Universal Robots PolyScope program: finalcoffee19-05-03.urp

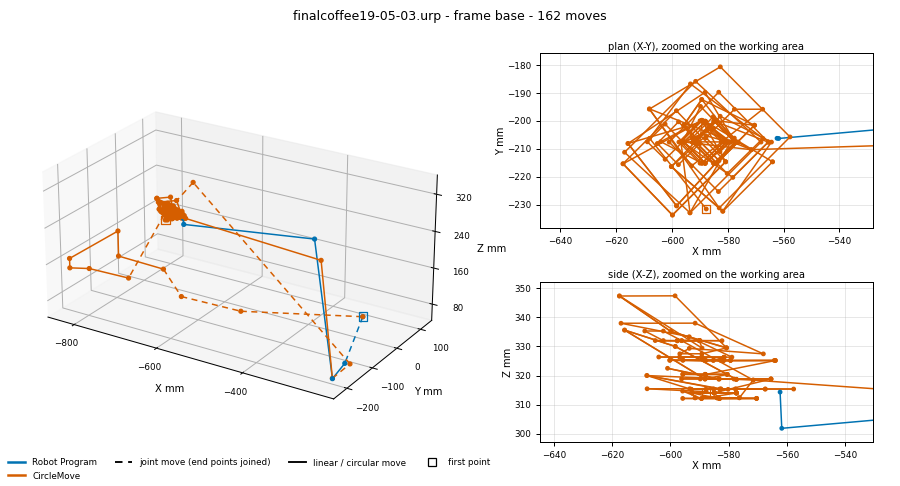
[picture p0: tool path of finalcoffee19-05-03.urp in frame base, 162 of 162 moves have a stored position in this frame; points joined in program order, loops and branches not executed]
Program finalcoffee19-05-03 (createdIn=3.3.3.292 lastSavedIn=3.3.3.292 directory=/programs/usbdisk_0 installation=default robotSerialNumber=2016353566)
Calibrated DH parameters: a=[0.000241, -0.028217, -0.285075, -0.000076, 0.000104, 0]; d=[0.089155, 574.834368, -342.811798, -231.912434, 0.094822, 0.082605]; alpha=[1.570306, 0.000738, 0.001161, 1.569845, -1.570892, 0]; deltaTheta=[0.000027, 1.504353, -0.747309, -0.757122, 0.000051, -0.000036]
Robot Program (runOnlyOnce=true motionType=MoveJ speed=1.047198 acceleration=1.396263 recalculateMotions=false)
  URCap com.ur.urcap.OnRobot.HelloWorldNode data=depthCompensate = false
    | width = 40
    | name = RG2(40)
    | force = 40
  MoveJ speed 20 deg/s, acceleration 30 deg/s^2 (recalculateMotions=false)
    Waypoint Waypoint_11: TCP in base x=-274.743 y=-2.169 z=93.833 mm, rx=1.4578 ry=-0.5495 rz=0.5386 rad; joints [-61.662, -71.825, 125.124, -50.852, -60.403, 38.941] deg; flange x=-270.843 y=184.262 z=86.813 mm, rx=1.4577 ry=-0.5495 rz=0.5386 rad
    Waypoint Waypoint_24: TCP in base x=-231.12 y=-150.401 z=66.269 mm, rx=0.5942 ry=1.8381 rz=-1.9212 rad; joints [-53.372, -80.21, 145.778, -62.89, -52.13, 33.023] deg; flange x=-227.221 y=36.081 z=59.238 mm, rx=1.4762 ry=-0.4771 rz=0.463 rad
  MoveP speed 76.2 mm/s, acceleration 1198.88 mm/s^2 (blendRadius=0.025 recalculateMotions=false) feature=Base
    Waypoint Waypoint_10: TCP in base x=-226.514 y=-206.056 z=58.912 mm, rx=0.3512 ry=2.0783 rz=-2.0466 rad; joints [-45.775, -85.681, 150.207, -66.123, -44.48, 19.129] deg; flange x=-222.338 y=-13.96 z=62.51 mm, rx=1.5718 ry=-0.2656 rz=0.2272 rad
  URCap com.ur.urcap.OnRobot.HelloWorldNode data=depthCompensate = false
    | width = 0
    | name = RG2(0)
    | force = 40
  URCap com.ur.urcap.OnRobot.TCPNode data=x = 5.6843418860808015E-14
    | y = -5.6843418860808015E-14
    | z = -2.5579538487363607E-13
    | rx = 0.0
    | ry = 5.551115123125783E-17
    | rz = 5.551115123125783E-17
    | xS = 0.0
    | yS = 0.0
    | zS = 0.0
    | rxS = 0.0
    | ryS = 0.0
    | rzS = 0.0
    | width = 40
    | tcpType = true
    | measuredWidthEnable = true
    | slaveSelected = false
    | TCP = TCP RG2()
  MoveL speed 76.2 mm/s, acceleration 254 mm/s^2 (recalculateMotions=false) feature=Base
    Waypoint wp_up: TCP in base x=-284.404 y=-181.482 z=326.495 mm, rx=0.3512 ry=2.0781 rz=-2.0466 rad; joints [-39.61, -106.093, 116.533, -12.17, -38.344, 19.314] deg; flange x=-280.343 y=5.056 z=329.988 mm, rx=1.5717 ry=-0.2657 rz=0.2273 rad
    Waypoint cup_center: TCP in base x=-561.773 y=-206.265 z=301.908 mm, rx=0.3623 ry=2.0424 rz=-1.9951 rad; joints [-18.068, -66.655, 77.97, -15.065, -18.801, 24.438] deg; flange x=-564.357 y=-14.16 z=305.939 mm, rx=1.5749 ry=-0.2793 rz=0.2941 rad
  MoveP speed 38.1 mm/s, acceleration 7.62 mm/s^2 (blendRadius=0.0127 recalculateMotions=false) feature=Base
    Waypoint cent_35: motionParameters(blendRadius=0.011); TCP in base x=-562.353 y=-206.199 z=314.344 mm, rx=0.5423 ry=1.9235 rz=-1.8764 rad; joints [-18.058, -66.887, 76.46, -13.315, -18.791, 35.8] deg; flange x=-564.912 y=-14.083 z=318.336 mm, rx=1.5494 ry=-0.4367 rz=0.4479 rad
    CircleMove
      Waypoint Waypoint_14: motionParameters(blendRadius=0.018); TCP in base x=-587.687 y=-231.512 z=314.467 mm, rx=0.5306 ry=1.932 rz=-1.8849 rad; joints [-14.904, -63.855, 72.029, -12.661, -15.633, 35.8] deg; flange x=-590.209 y=-39.4 z=318.513 mm, rx=1.5515 ry=-0.4261 rz=0.4373 rad
      Waypoint deg_left_36: motionParameters(blendRadius=0.013); TCP in base x=-607.977 y=-206.219 z=315.477 mm, rx=0.5411 ry=1.9244 rz=-1.8774 rad; joints [-16.716, -60.481, 66.783, -10.318, -17.442, 36.007] deg; flange x=-610.544 y=-14.142 z=319.49 mm, rx=1.5496 ry=-0.4357 rz=0.4467 rad
  MoveP speed 25.4 mm/s, acceleration 76.2 mm/s^2 (blendRadius=0.00635 recalculateMotions=false) feature=Base
    CircleMove
      Waypoint Waypoint_120: motionParameters(blendRadius=0.011); TCP in base x=-593.35 y=-186.719 z=315.478 mm, rx=0.5524 ry=1.9162 rz=-1.8691 rad; joints [-18.922, -62.136, 69.295, -10.741, -19.654, 36.3] deg; flange x=-595.922 y=5.421 z=319.508 mm, rx=1.5475 ry=-0.446 rz=0.457 rad
      Waypoint Waypoint_121: motionParameters(blendRadius=0.006); TCP in base x=-567.406 y=-206.241 z=315.399 mm, rx=0.5493 ry=1.9185 rz=-1.8715 rad; joints [-17.897, -66.224, 75.343, -12.894, -18.625, 36.3] deg; flange x=-569.935 y=-14.123 z=319.455 mm, rx=1.5481 ry=-0.4432 rz=0.4541 rad
    CircleMove
      Waypoint Waypoint_122: motionParameters(blendRadius=0.01); TCP in base x=-580.202 y=-218.815 z=315.281 mm, rx=0.5491 ry=1.9188 rz=-1.8724 rad; joints [-16.313, -64.705, 73.156, -12.546, -17.023, 36.581] deg; flange x=-582.655 y=-26.726 z=319.337 mm, rx=1.548 ry=-0.4427 rz=0.4531 rad
      Waypoint Waypoint_123: motionParameters(blendRadius=0.006); TCP in base x=-592.797 y=-206.153 z=315.297 mm, rx=0.5517 ry=1.9167 rz=-1.87 rad; joints [-17.153, -62.662, 70.126, -11.364, -17.868, 36.6] deg; flange x=-595.328 y=-13.997 z=319.293 mm, rx=1.5474 ry=-0.4457 rz=0.4562 rad
    CircleMove
      Waypoint Waypoint_124: motionParameters(blendRadius=0.003); TCP in base x=-585.199 y=-198.492 z=315.45 mm, rx=0.5527 ry=1.916 rz=-1.869 rad; joints [-18.086, -63.573, 71.462, -11.621, -18.81, 36.485] deg; flange x=-587.756 y=-6.367 z=319.434 mm, rx=1.5474 ry=-0.4464 rz=0.4572 rad
      Waypoint Waypoint_125: motionParameters(blendRadius=0.003); TCP in base x=-577.639 y=-206.134 z=315.376 mm, rx=0.5537 ry=1.9154 rz=-1.8684 rad; joints [-17.596, -64.801, 73.285, -12.319, -18.315, 36.654] deg; flange x=-580.185 y=-13.996 z=319.379 mm, rx=1.5472 ry=-0.4474 rz=0.4579 rad
    MoveP speed 25.4 mm/s, acceleration 25.4 mm/s^2 (blendRadius=0.00508 recalculateMotions=false) feature=Base
      CircleMove
        Waypoint Waypoint_3: motionParameters(blendRadius=0.001); TCP in base x=-582.779 y=-210.988 z=315.338 mm, rx=0.5617 ry=1.9099 rz=-1.8632 rad; joints [-16.989, -64.197, 72.405, -12.165, -17.686, 37.3] deg; flange x=-585.236 y=-18.851 z=319.337 mm, rx=1.5456 ry=-0.4548 rz=0.4646 rad
        Waypoint cen_l_7: motionParameters(blendRadius=0.005); TCP in base x=-587.786 y=-206 z=315.362 mm, rx=0.5628 ry=1.9089 rz=-1.8623 rad; joints [-17.305, -63.384, 71.194, -11.692, -18.016, 37.3] deg; flange x=-590.262 y=-13.929 z=319.365 mm, rx=1.5454 ry=-0.4557 rz=0.4659 rad
    MoveP speed 33.02 mm/s, acceleration 76.2 mm/s^2 (blendRadius=0.00762 recalculateMotions=false) feature=Base
      CircleMove
        Waypoint Waypoint_2: motionParameters(blendRadius=0.008); TCP in base x=-577.621 y=-195.808 z=315.417 mm, rx=0.5695 ry=1.9041 rz=-1.8572 rad; joints [-18.573, -64.59, 72.957, -12.025, -19.283, 37.5] deg; flange x=-580.119 y=-3.7 z=319.475 mm, rx=1.5442 ry=-0.4618 rz=0.4718 rad
        Waypoint Waypoint_5: motionParameters(blendRadius=0.001); TCP in base x=-567.485 y=-195.794 z=315.362 mm, rx=0.5701 ry=1.9035 rz=-1.8567 rad; joints [-18.9, -65.989, 75.013, -12.613, -19.611, 37.5] deg; flange x=-569.984 y=-3.689 z=319.375 mm, rx=1.544 ry=-0.4627 rz=0.4728 rad
      CircleMove
        Waypoint Waypoint_6: motionParameters(blendRadius=0.017); TCP in base x=-592.923 y=-216.078 z=315.3 mm, rx=0.5649 ry=1.9075 rz=-1.8608 rad; joints [-16.226, -62.864, 70.427, -11.703, -16.927, 37.7] deg; flange x=-595.396 y=-23.94 z=319.322 mm, rx=1.545 ry=-0.4577 rz=0.4675 rad
        Waypoint Waypoint_8: motionParameters(blendRadius=0.007); TCP in base x=-608.08 y=-195.76 z=320.03 mm, rx=0.5712 ry=1.9029 rz=-1.8561 rad; joints [-17.668, -60.32, 65.859, -9.368, -18.376, 37.8] deg; flange x=-610.553 y=-3.603 z=324.066 mm, rx=1.5439 ry=-0.4635 rz=0.4733 rad
      CircleMove
        Waypoint Waypoint_126: motionParameters(blendRadius=0.021); TCP in base x=-582.652 y=-180.614 z=315.453 mm, rx=0.5799 ry=1.8963 rz=-1.8492 rad; joints [-19.829, -63.501, 71.344, -11.288, -20.55, 38] deg; flange x=-585.205 y=11.524 z=319.472 mm, rx=1.5422 ry=-0.4716 rz=0.4818 rad
        Waypoint Waypoint_9: motionParameters(jointSpeed=1.047198 jointAcceleration=1.396263 cartesianSpeed=0.0381 cartesianAcceleration=0.0254 blendRadius=0.014); TCP in base x=-557.692 y=-205.719 z=315.384 mm, rx=0.5784 ry=1.8973 rz=-1.8503 rad; joints [-18.254, -67.548, 77.238, -13.406, -18.985, 38.191] deg; flange x=-560.213 y=-13.613 z=319.44 mm, rx=1.5425 ry=-0.4702 rz=0.4805 rad
      CircleMove
        Waypoint Waypoint_37: motionParameters(jointSpeed=1.047198 jointAcceleration=1.396263 cartesianSpeed=0.01778 cartesianAcceleration=0.0254 blendRadius=0.020005); TCP in base x=-583.059 y=-231.133 z=315.374 mm, rx=0.5791 ry=1.8967 rz=-1.8497 rad; joints [-15.057, -64.504, 72.861, -12.792, -15.796, 39] deg; flange x=-585.632 y=-39.012 z=319.369 mm, rx=1.5423 ry=-0.4709 rz=0.4813 rad
        Waypoint Waypoint_36: motionParameters(jointSpeed=1.047198 jointAcceleration=1.396263 cartesianSpeed=0.0254 cartesianAcceleration=0.0254); TCP in base x=-608.023 y=-195.66 z=320.009 mm, rx=0.5826 ry=1.8944 rz=-1.8475 rad; joints [-17.674, -60.321, 65.86, -9.366, -18.383, 38.578] deg; flange x=-610.535 y=-3.547 z=324.069 mm, rx=1.5416 ry=-0.4742 rz=0.4839 rad
  'bloom finished'
  MoveL speed 76.2 mm/s, acceleration 635 mm/s^2 (recalculateMotions=false) feature=Base
    Waypoint cup_cent: TCP in base x=-571.578 y=-210.276 z=318.459 mm, rx=0.4644 ry=1.9797 rz=-1.9328 rad; joints [-17.399, -65.896, 74.417, -12.484, -18.002, 30.817] deg; flange x=-573.709 y=-18.152 z=322.504 mm, rx=1.5623 ry=-0.3665 rz=0.3757 rad
  Wait Sleep waitTime=29
  'first_pour'
  MoveP speed 12.7 mm/s, acceleration 10.16 mm/s^2 (blendRadius=0.00762 recalculateMotions=false) feature=Base
    Waypoint cent_39: motionParameters(jointSpeed=1.047198 jointAcceleration=1.396263 cartesianSpeed=0.0254 cartesianAcceleration=0.0508 blendRadius=0); TCP in base x=-576.315 y=-207.596 z=312.389 mm, rx=0.5992 ry=1.8838 rz=-1.8375 rad; joints [-17.511, -65.048, 74.074, -12.957, -18.124, 39.682] deg; flange x=-578.469 y=-15.487 z=316.479 mm, rx=1.5382 ry=-0.4894 rz=0.496 rad
    Loop Counting (count=1) loopVariable(name=Loop_1)
      MoveP speed 25.4 mm/s, acceleration 10.16 mm/s^2 (blendRadius=0.00762 recalculateMotions=false) feature=Base
        CircleMove
          Waypoint Waypoint_7: TCP in base x=-583.932 y=-215.142 z=312.393 mm, rx=0.5993 ry=1.8838 rz=-1.8376 rad; joints [-16.567, -64.138, 72.741, -12.744, -17.183, 39.898] deg; flange x=-586.097 y=-23.083 z=316.469 mm, rx=1.5383 ry=-0.4893 rz=0.4959 rad
          Waypoint Waypoint_26: TCP in base x=-591.514 y=-207.599 z=312.378 mm, rx=0.5991 ry=1.8838 rz=-1.8375 rad; joints [-17.067, -62.917, 70.922, -12.035, -17.686, 39.778] deg; flange x=-593.69 y=-15.47 z=316.465 mm, rx=1.5383 ry=-0.4892 rz=0.4959 rad
        CircleMove
          Waypoint Waypoint_27: TCP in base x=-583.922 y=-199.93 z=312.363 mm, rx=0.5993 ry=1.8837 rz=-1.8376 rad; joints [-18.004, -63.821, 72.265, -12.276, -18.612, 39.567] deg; flange x=-586.103 y=-7.836 z=316.474 mm, rx=1.5383 ry=-0.4893 rz=0.4958 rad
          Waypoint Waypoint_28: TCP in base x=-576.335 y=-207.56 z=312.393 mm, rx=0.5992 ry=1.8838 rz=-1.8376 rad; joints [-17.512, -65.047, 74.074, -12.96, -18.125, 39.678] deg; flange x=-578.474 y=-15.472 z=316.467 mm, rx=1.5383 ry=-0.4893 rz=0.4959 rad
    MoveP speed 25.4 mm/s, acceleration 7.62 mm/s^2 (blendRadius=0.00762 recalculateMotions=false) feature=Base
      CircleMove
        Waypoint Waypoint_29: TCP in base x=-583.932 y=-215.142 z=312.393 mm, rx=0.5993 ry=1.8838 rz=-1.8376 rad; joints [-16.567, -64.138, 72.741, -12.744, -17.183, 39.898] deg; flange x=-586.097 y=-23.083 z=316.469 mm, rx=1.5383 ry=-0.4893 rz=0.4959 rad
        Waypoint Waypoint_30: TCP in base x=-591.514 y=-207.599 z=312.378 mm, rx=0.5991 ry=1.8838 rz=-1.8375 rad; joints [-17.067, -62.917, 70.922, -12.035, -17.686, 39.778] deg; flange x=-593.69 y=-15.47 z=316.465 mm, rx=1.5383 ry=-0.4892 rz=0.4959 rad
      CircleMove
        Waypoint Waypoint_31: motionParameters(blendRadius=0.002997); TCP in base x=-583.922 y=-199.93 z=312.363 mm, rx=0.5993 ry=1.8837 rz=-1.8376 rad; joints [-18.004, -63.821, 72.265, -12.276, -18.612, 39.567] deg; flange x=-586.103 y=-7.836 z=316.474 mm, rx=1.5383 ry=-0.4893 rz=0.4958 rad
        Waypoint next40: motionParameters(jointSpeed=1.047198 jointAcceleration=1.396263 cartesianSpeed=0.01778 cartesianAcceleration=0.0254); TCP in base x=-570.424 y=-201.531 z=312.179 mm, rx=0.6107 ry=1.875 rz=-1.8287 rad; joints [-18.272, -65.726, 75.088, -13.146, -18.889, 40.324] deg; flange x=-572.598 y=-9.409 z=316.276 mm, rx=1.5358 ry=-0.5003 rz=0.5068 rad
    Waypoint cent_40: motionParameters(blendRadius=0); TCP in base x=-570.415 y=-201.533 z=312.191 mm, rx=0.6107 ry=1.875 rz=-1.8286 rad; joints [-18.272, -65.726, 75.088, -13.146, -18.889, 40.324] deg; flange x=-572.598 y=-9.409 z=316.276 mm, rx=1.5358 ry=-0.5003 rz=0.5068 rad
    Loop Counting (count=1) loopVariable(name=Loop_2)
      MoveP speed 25.4 mm/s, acceleration 7.62 mm/s^2 (blendRadius=0.0127 recalculateMotions=false) feature=Base
        CircleMove
          Waypoint Waypoint_32: TCP in base x=-583.144 y=-214.174 z=312.098 mm, rx=0.611 ry=1.8748 rz=-1.8286 rad; joints [-16.683, -64.226, 72.9, -12.797, -17.304, 40.678] deg; flange x=-585.307 y=-22.093 z=316.257 mm, rx=1.5358 ry=-0.5003 rz=0.5068 rad
          Waypoint Waypoint_33: TCP in base x=-595.764 y=-201.544 z=312.163 mm, rx=0.6107 ry=1.875 rz=-1.8286 rad; joints [-17.505, -62.173, 69.832, -11.602, -18.129, 40.488] deg; flange x=-597.992 y=-9.403 z=316.253 mm, rx=1.5359 ry=-0.5002 rz=0.5068 rad
        CircleMove
          Waypoint Waypoint_34: TCP in base x=-589.315 y=-192.31 z=312.12 mm, rx=0.6107 ry=1.8749 rz=-1.8284 rad; joints [-18.55, -62.88, 70.893, -11.747, -19.173, 40.274] deg; flange x=-591.505 y=-0.185 z=316.249 mm, rx=1.5359 ry=-0.5003 rz=0.5069 rad
          Waypoint Waypoint_35: TCP in base x=-570.432 y=-201.519 z=312.152 mm, rx=0.6108 ry=1.875 rz=-1.8286 rad; joints [-18.272, -65.726, 75.088, -13.151, -18.892, 40.328] deg; flange x=-572.601 y=-9.409 z=316.281 mm, rx=1.5359 ry=-0.5003 rz=0.5068 rad
    MoveP speed 25.4 mm/s, acceleration 7.62 mm/s^2 (blendRadius=0.0127 recalculateMotions=false) feature=Base
      CircleMove
        Waypoint Waypoint_32: TCP in base x=-583.144 y=-214.174 z=312.098 mm, rx=0.611 ry=1.8748 rz=-1.8286 rad; joints [-16.683, -64.226, 72.9, -12.797, -17.304, 40.678] deg; flange x=-585.307 y=-22.093 z=316.257 mm, rx=1.5358 ry=-0.5003 rz=0.5068 rad
        Waypoint bts_mid_40: TCP in base x=-595.797 y=-201.584 z=314.675 mm, rx=0.6105 ry=1.8753 rz=-1.8286 rad; joints [-17.503, -62.219, 69.536, -11.27, -18.121, 40.493] deg; flange x=-598.023 y=-9.423 z=318.729 mm, rx=1.5359 ry=-0.5002 rz=0.5067 rad
      CircleMove
        Waypoint bts_Waypoint_34: TCP in base x=-589.305 y=-192.307 z=312.113 mm, rx=0.6107 ry=1.8749 rz=-1.8284 rad; joints [-18.548, -62.875, 70.89, -11.75, -19.176, 40.276] deg; flange x=-591.532 y=-0.186 z=316.211 mm, rx=1.5359 ry=-0.5002 rz=0.507 rad
        Waypoint bts_41: TCP in base x=-577.315 y=-207.686 z=314.026 mm, rx=0.6254 ry=1.8636 rz=-1.8173 rad; joints [-17.476, -64.94, 73.67, -12.672, -18.095, 41.504] deg; flange x=-579.514 y=-15.524 z=318.136 mm, rx=1.5325 ry=-0.5143 rz=0.5204 rad
    Waypoint cent_41: motionParameters(blendRadius=0); TCP in base x=-577.334 y=-207.648 z=314.054 mm, rx=0.6254 ry=1.8638 rz=-1.8175 rad; joints [-17.478, -64.943, 73.67, -12.67, -18.097, 41.506] deg; flange x=-579.495 y=-15.499 z=318.162 mm, rx=1.5325 ry=-0.5143 rz=0.5204 rad
    Loop Counting (count=1) loopVariable(name=Loop_3)
      MoveP speed 25.4 mm/s, acceleration 10.16 mm/s^2 (blendRadius=0.00762 recalculateMotions=false) feature=Base
        CircleMove
          Waypoint Waypoint_39: TCP in base x=-584.951 y=-215.263 z=314.085 mm, rx=0.6254 ry=1.8638 rz=-1.8176 rad; joints [-16.532, -64.028, 72.332, -12.453, -17.154, 41.721] deg; flange x=-587.132 y=-23.144 z=318.13 mm, rx=1.5325 ry=-0.5142 rz=0.5204 rad
          Waypoint Waypoint_40: TCP in base x=-592.538 y=-207.689 z=314.112 mm, rx=0.6252 ry=1.8639 rz=-1.8175 rad; joints [-17.03, -62.803, 70.499, -11.737, -17.657, 41.607] deg; flange x=-594.735 y=-15.541 z=318.178 mm, rx=1.5326 ry=-0.5142 rz=0.5205 rad
        CircleMove
          Waypoint Waypoint_41: TCP in base x=-584.885 y=-200.048 z=314.03 mm, rx=0.6252 ry=1.8638 rz=-1.8174 rad; joints [-17.966, -63.709, 71.859, -11.99, -18.591, 41.396] deg; flange x=-587.129 y=-7.902 z=318.092 mm, rx=1.5326 ry=-0.5142 rz=0.5205 rad
          Waypoint Waypoint_42: TCP in base x=-577.306 y=-207.68 z=314.014 mm, rx=0.6253 ry=1.8637 rz=-1.8174 rad; joints [-17.476, -64.94, 73.67, -12.672, -18.095, 41.504] deg; flange x=-579.514 y=-15.524 z=318.136 mm, rx=1.5325 ry=-0.5143 rz=0.5204 rad
    MoveP speed 25.4 mm/s, acceleration 7.62 mm/s^2 (blendRadius=0.00762 recalculateMotions=false) feature=Base
      CircleMove
        Waypoint Waypoint_43: TCP in base x=-584.951 y=-215.263 z=314.085 mm, rx=0.6254 ry=1.8638 rz=-1.8176 rad; joints [-16.532, -64.028, 72.332, -12.453, -17.154, 41.721] deg; flange x=-587.132 y=-23.144 z=318.13 mm, rx=1.5325 ry=-0.5142 rz=0.5204 rad
        Waypoint Waypoint_44: TCP in base x=-592.538 y=-207.689 z=314.112 mm, rx=0.6252 ry=1.8639 rz=-1.8175 rad; joints [-17.03, -62.803, 70.499, -11.737, -17.657, 41.607] deg; flange x=-594.735 y=-15.541 z=318.178 mm, rx=1.5326 ry=-0.5142 rz=0.5205 rad
      CircleMove
        Waypoint Waypoint_45: motionParameters(blendRadius=0.002); TCP in base x=-584.885 y=-200.048 z=314.03 mm, rx=0.6252 ry=1.8638 rz=-1.8174 rad; joints [-17.966, -63.709, 71.859, -11.99, -18.591, 41.396] deg; flange x=-587.129 y=-7.902 z=318.092 mm, rx=1.5326 ry=-0.5142 rz=0.5205 rad
        Waypoint next_42: motionParameters(jointSpeed=1.047198 jointAcceleration=1.396263 cartesianSpeed=0.01778 cartesianAcceleration=0.0254); TCP in base x=-577.322 y=-207.657 z=314.049 mm, rx=0.6398 ry=1.8525 rz=-1.8063 rad; joints [-17.476, -64.94, 73.671, -12.668, -18.093, 42.507] deg; flange x=-579.505 y=-15.524 z=318.13 mm, rx=1.5292 ry=-0.5282 rz=0.534 rad
    Waypoint cent_42: motionParameters(blendRadius=0); TCP in base x=-577.341 y=-207.607 z=314.023 mm, rx=0.6399 ry=1.8525 rz=-1.8064 rad; joints [-17.478, -64.938, 73.671, -12.671, -18.097, 42.506] deg; flange x=-579.514 y=-15.502 z=318.108 mm, rx=1.5292 ry=-0.5281 rz=0.534 rad
    Loop Counting (count=1) loopVariable(name=Loop_4)
      MoveP speed 25.4 mm/s, acceleration 7.62 mm/s^2 (blendRadius=0.00762 recalculateMotions=false) feature=Base
        CircleMove
          Waypoint Waypoint_46: TCP in base x=-584.946 y=-215.223 z=314.082 mm, rx=0.6398 ry=1.8526 rz=-1.8065 rad; joints [-16.533, -64.029, 72.333, -12.455, -17.154, 42.725] deg; flange x=-587.131 y=-23.131 z=318.132 mm, rx=1.5292 ry=-0.5281 rz=0.5339 rad
          Waypoint Waypoint_47: TCP in base x=-592.537 y=-207.645 z=314.048 mm, rx=0.6397 ry=1.8525 rz=-1.8063 rad; joints [-17.031, -62.802, 70.499, -11.736, -17.651, 42.609] deg; flange x=-594.75 y=-15.528 z=318.16 mm, rx=1.5292 ry=-0.5281 rz=0.5339 rad
        CircleMove
          Waypoint Waypoint_48: TCP in base x=-584.912 y=-200.025 z=314.093 mm, rx=0.6396 ry=1.8527 rz=-1.8064 rad; joints [-17.966, -63.713, 71.855, -11.981, -18.586, 42.402] deg; flange x=-587.118 y=-7.901 z=318.164 mm, rx=1.5292 ry=-0.5281 rz=0.534 rad
          Waypoint Waypoint_49: TCP in base x=-577.321 y=-207.614 z=314.06 mm, rx=0.6398 ry=1.8526 rz=-1.8065 rad; joints [-17.48, -64.938, 73.672, -12.671, -18.096, 42.506] deg; flange x=-579.512 y=-15.482 z=318.099 mm, rx=1.5292 ry=-0.5282 rz=0.534 rad
    MoveP speed 25.4 mm/s, acceleration 7.62 mm/s^2 (blendRadius=0.00762 recalculateMotions=false) feature=Base
      CircleMove
        Waypoint Waypoint_50: TCP in base x=-584.946 y=-215.223 z=314.082 mm, rx=0.6398 ry=1.8526 rz=-1.8065 rad; joints [-16.533, -64.029, 72.333, -12.455, -17.154, 42.725] deg; flange x=-587.131 y=-23.131 z=318.132 mm, rx=1.5292 ry=-0.5281 rz=0.5339 rad
        Waypoint Waypoint_51: TCP in base x=-592.537 y=-207.645 z=314.048 mm, rx=0.6397 ry=1.8525 rz=-1.8063 rad; joints [-17.031, -62.802, 70.499, -11.736, -17.651, 42.609] deg; flange x=-594.75 y=-15.528 z=318.16 mm, rx=1.5292 ry=-0.5281 rz=0.5339 rad
      CircleMove
        Waypoint Waypoint_52: TCP in base x=-584.912 y=-200.025 z=314.093 mm, rx=0.6396 ry=1.8527 rz=-1.8064 rad; joints [-17.966, -63.713, 71.855, -11.981, -18.586, 42.402] deg; flange x=-587.118 y=-7.901 z=318.164 mm, rx=1.5292 ry=-0.5281 rz=0.534 rad
        Waypoint next_43: motionParameters(jointSpeed=1.047198 jointAcceleration=1.396263 cartesianSpeed=0.01778 cartesianAcceleration=0.0254); TCP in base x=-565.488 y=-207.564 z=318.804 mm, rx=0.6541 ry=1.8415 rz=-1.7955 rad; joints [-17.845, -66.686, 75.497, -12.68, -18.459, 43.426] deg; flange x=-567.635 y=-15.452 z=322.878 mm, rx=1.5258 ry=-0.5419 rz=0.5473 rad
    Waypoint cent43: motionParameters(blendRadius=0); TCP in base x=-565.48 y=-207.533 z=318.836 mm, rx=0.654 ry=1.8416 rz=-1.7955 rad; joints [-17.848, -66.685, 75.498, -12.68, -18.455, 43.427] deg; flange x=-567.641 y=-15.422 z=322.875 mm, rx=1.5257 ry=-0.542 rz=0.5472 rad
    Loop Counting (count=1) loopVariable(name=Loop_5)
      MoveP speed 25.4 mm/s, acceleration 7.62 mm/s^2 (blendRadius=0.01778 recalculateMotions=false) feature=Base
        CircleMove
          Waypoint Waypoint_53: motionParameters(blendRadius=0.016); TCP in base x=-583.332 y=-225.271 z=318.734 mm, rx=0.6464 ry=1.8476 rz=-1.8017 rad; joints [-15.628, -64.549, 72.413, -12.234, -16.234, 43.4] deg; flange x=-585.428 y=-33.151 z=322.819 mm, rx=1.5276 ry=-0.5344 rz=0.5397 rad
          Waypoint Waypoint_54: motionParameters(blendRadius=0.008); TCP in base x=-600.969 y=-207.565 z=322.496 mm, rx=0.6537 ry=1.8418 rz=-1.7954 rad; joints [-16.806, -61.741, 67.661, -10.03, -17.424, 43.663] deg; flange x=-603.173 y=-15.419 z=326.573 mm, rx=1.526 ry=-0.5417 rz=0.5471 rad
        CircleMove
          Waypoint Waypoint_55: motionParameters(blendRadius=0.016); TCP in base x=-583.224 y=-189.699 z=318.906 mm, rx=0.6567 ry=1.8396 rz=-1.7933 rad; joints [-18.984, -63.819, 71.288, -11.149, -19.592, 43.4] deg; flange x=-585.391 y=2.423 z=323.037 mm, rx=1.5253 ry=-0.5444 rz=0.5496 rad
          Waypoint Waypoint_56: motionParameters(blendRadius=0.007); TCP in base x=-565.473 y=-207.549 z=318.864 mm, rx=0.6538 ry=1.8418 rz=-1.7956 rad; joints [-17.849, -66.69, 75.494, -12.685, -18.462, 43.43] deg; flange x=-567.633 y=-15.408 z=322.934 mm, rx=1.5259 ry=-0.5418 rz=0.5471 rad
    MoveP speed 25.4 mm/s, acceleration 12.7 mm/s^2 (blendRadius=0.0127 recalculateMotions=false) feature=Base
      CircleMove
        Waypoint Waypoint_57: motionParameters(blendRadius=0.009); TCP in base x=-578.173 y=-220.21 z=318.818 mm, rx=0.6539 ry=1.8417 rz=-1.7956 rad; joints [-16.247, -65.181, 73.313, -12.375, -16.865, 43.798] deg; flange x=-580.319 y=-28.132 z=322.966 mm, rx=1.526 ry=-0.5417 rz=0.547 rad
        Waypoint Waypoint_58: motionParameters(blendRadius=0.008); TCP in base x=-596.136 y=-207.498 z=318.857 mm, rx=0.654 ry=1.8416 rz=-1.7954 rad; joints [-16.941, -62.382, 69.164, -10.847, -17.558, 43.631] deg; flange x=-598.3 y=-15.422 z=322.939 mm, rx=1.5258 ry=-0.5419 rz=0.5473 rad
      CircleMove
        Waypoint Waypoint_59: motionParameters(blendRadius=0.005); TCP in base x=-589.749 y=-194.774 z=318.845 mm, rx=0.654 ry=1.8417 rz=-1.7956 rad; joints [-18.314, -63.017, 70.113, -10.888, -18.915, 43.329] deg; flange x=-591.889 y=-2.613 z=322.931 mm, rx=1.5259 ry=-0.5419 rz=0.5469 rad
        Waypoint btsnext_44: motionParameters(jointSpeed=1.047198 jointAcceleration=1.396263 cartesianSpeed=0.01778 cartesianAcceleration=0.0254); TCP in base x=-577.378 y=-207.588 z=318.721 mm, rx=0.6682 ry=1.8298 rz=-1.7838 rad; joints [-17.473, -65.02, 73.092, -12.001, -18.108, 44.514] deg; flange x=-579.589 y=-15.517 z=322.84 mm, rx=1.5223 ry=-0.5557 rz=0.5613 rad
    Waypoint cent_44: motionParameters(blendRadius=0); TCP in base x=-577.37 y=-207.623 z=318.709 mm, rx=0.6681 ry=1.8298 rz=-1.7838 rad; joints [-17.473, -65.02, 73.092, -12.001, -18.108, 44.514] deg; flange x=-579.589 y=-15.517 z=322.84 mm, rx=1.5223 ry=-0.5557 rz=0.5613 rad
    Loop Counting (count=1) loopVariable(name=Loop_6)
      MoveP speed 25.4 mm/s, acceleration 12.7 mm/s^2 (blendRadius=0.00762 recalculateMotions=false) feature=Base
        CircleMove
          Waypoint Waypoint_60: TCP in base x=-598.311 y=-230.402 z=329.993 mm, rx=0.6681 ry=1.8301 rz=-1.784 rad; joints [-14.756, -62.667, 67.963, -9.907, -15.391, 45.214] deg; flange x=-600.502 y=-38.296 z=334.104 mm, rx=1.5224 ry=-0.5556 rz=0.561 rad
          Waypoint Waypoint_61: TCP in base x=-615.716 y=-208.072 z=335.618 mm, rx=0.668 ry=1.83 rz=-1.7839 rad; joints [-16.359, -59.704, 62.616, -7.089, -16.997, 44.767] deg; flange x=-617.929 y=-15.958 z=339.722 mm, rx=1.5224 ry=-0.5556 rz=0.5612 rad
        CircleMove
          Waypoint Waypoint_62: TCP in base x=-588.125 y=-189.74 z=318.812 mm, rx=0.6678 ry=1.8303 rz=-1.7841 rad; joints [-18.817, -63.11, 70.256, -10.833, -19.449, 44.231] deg; flange x=-590.331 y=2.32 z=322.895 mm, rx=1.5225 ry=-0.5554 rz=0.5609 rad
          Waypoint Waypoint_63: TCP in base x=-577.371 y=-207.629 z=318.712 mm, rx=0.6681 ry=1.8298 rz=-1.7838 rad; joints [-17.473, -65.02, 73.092, -12.001, -18.108, 44.514] deg; flange x=-579.589 y=-15.517 z=322.84 mm, rx=1.5223 ry=-0.5557 rz=0.5613 rad
    MoveP speed 25.4 mm/s, acceleration 12.7 mm/s^2 (blendRadius=0.00762 recalculateMotions=false) feature=Base
      CircleMove
        Waypoint Waypoint_64: TCP in base x=-598.327 y=-230.375 z=330.025 mm, rx=0.6682 ry=1.8301 rz=-1.784 rad; joints [-14.758, -62.665, 67.963, -9.906, -15.391, 45.215] deg; flange x=-600.511 y=-38.278 z=334.075 mm, rx=1.5223 ry=-0.5557 rz=0.5611 rad
        Waypoint Waypoint_65: TCP in base x=-615.696 y=-208.061 z=335.611 mm, rx=0.668 ry=1.8299 rz=-1.7838 rad; joints [-16.359, -59.701, 62.616, -7.088, -16.996, 44.767] deg; flange x=-617.943 y=-15.948 z=339.696 mm, rx=1.5223 ry=-0.5557 rz=0.5612 rad
      CircleMove
        Waypoint Waypoint_66: TCP in base x=-588.085 y=-200.014 z=318.836 mm, rx=0.6677 ry=1.8303 rz=-1.784 rad; joints [-17.874, -63.347, 70.611, -11.132, -18.502, 44.419] deg; flange x=-590.351 y=-7.845 z=322.91 mm, rx=1.5225 ry=-0.5554 rz=0.5608 rad
        Waypoint next_45: motionParameters(jointSpeed=1.047198 jointAcceleration=1.396263 cartesianSpeed=0.01778 cartesianAcceleration=0.0254); TCP in base x=-580.527 y=-207.539 z=320.413 mm, rx=0.6803 ry=1.8202 rz=-1.7743 rad; joints [-17.388, -64.612, 72.255, -11.595, -18.015, 45.402] deg; flange x=-582.732 y=-15.437 z=324.471 mm, rx=1.5192 ry=-0.5677 rz=0.5728 rad
    Waypoint cent_45: motionParameters(blendRadius=0); TCP in base x=-580.529 y=-207.561 z=320.393 mm, rx=0.6802 ry=1.8202 rz=-1.7743 rad; joints [-17.383, -64.612, 72.256, -11.591, -18.016, 45.399] deg; flange x=-582.722 y=-15.488 z=324.463 mm, rx=1.5192 ry=-0.5676 rz=0.5729 rad
    Loop Counting (count=1) loopVariable(name=Loop_7)
      MoveP speed 25.4 mm/s, acceleration 14.99 mm/s^2 (blendRadius=0.00762 recalculateMotions=false) feature=Base
        CircleMove
          Waypoint Waypoint_67: TCP in base x=-588.078 y=-215.151 z=320.442 mm, rx=0.6803 ry=1.8201 rz=-1.7743 rad; joints [-16.449, -63.693, 70.9, -11.369, -17.081, 45.617] deg; flange x=-590.337 y=-23.067 z=324.482 mm, rx=1.5192 ry=-0.5676 rz=0.5727 rad
          Waypoint Waypoint_68: TCP in base x=-595.729 y=-207.551 z=320.45 mm, rx=0.68 ry=1.8204 rz=-1.7743 rad; joints [-16.947, -62.453, 69.038, -10.642, -17.578, 45.501] deg; flange x=-597.967 y=-15.458 z=324.52 mm, rx=1.5193 ry=-0.5675 rz=0.5727 rad
        CircleMove
          Waypoint Waypoint_69: TCP in base x=-587.953 y=-200.162 z=320.371 mm, rx=0.6801 ry=1.8202 rz=-1.7743 rad; joints [-17.863, -63.405, 70.471, -10.917, -18.495, 45.295] deg; flange x=-590.13 y=-8.029 z=324.446 mm, rx=1.5192 ry=-0.5676 rz=0.5729 rad
          Waypoint Waypoint_70: TCP in base x=-580.495 y=-207.606 z=320.417 mm, rx=0.68 ry=1.8204 rz=-1.7743 rad; joints [-17.388, -64.612, 72.255, -11.595, -18.015, 45.402] deg; flange x=-582.732 y=-15.437 z=324.471 mm, rx=1.5192 ry=-0.5677 rz=0.5728 rad
    MoveP speed 25.4 mm/s, acceleration 12.7 mm/s^2 (blendRadius=0.00762 recalculateMotions=false) feature=Base
      CircleMove
        Waypoint Waypoint_71: TCP in base x=-588.078 y=-215.151 z=320.442 mm, rx=0.6803 ry=1.8201 rz=-1.7743 rad; joints [-16.449, -63.693, 70.9, -11.369, -17.081, 45.617] deg; flange x=-590.337 y=-23.067 z=324.482 mm, rx=1.5192 ry=-0.5676 rz=0.5727 rad
        Waypoint Waypoint_72: TCP in base x=-595.729 y=-207.551 z=320.45 mm, rx=0.68 ry=1.8204 rz=-1.7743 rad; joints [-16.947, -62.453, 69.038, -10.642, -17.578, 45.501] deg; flange x=-597.967 y=-15.458 z=324.52 mm, rx=1.5193 ry=-0.5675 rz=0.5727 rad
      CircleMove
        Waypoint Waypoint_73: TCP in base x=-587.953 y=-200.162 z=320.371 mm, rx=0.6801 ry=1.8202 rz=-1.7743 rad; joints [-17.863, -63.405, 70.471, -10.917, -18.495, 45.295] deg; flange x=-590.13 y=-8.029 z=324.446 mm, rx=1.5192 ry=-0.5676 rz=0.5729 rad
        Waypoint next_46: TCP in base x=-563.961 y=-214.615 z=325.18 mm, rx=0.695 ry=1.808 rz=-1.7618 rad; joints [-17.2, -67.152, 75.219, -12.074, -17.843, 46.553] deg; flange x=-566.211 y=-22.508 z=329.281 mm, rx=1.5153 ry=-0.5826 rz=0.5877 rad
    Waypoint cent_46: motionParameters(blendRadius=0); TCP in base x=-563.961 y=-214.631 z=325.185 mm, rx=0.6951 ry=1.8079 rz=-1.7617 rad; joints [-17.2, -67.151, 75.221, -12.07, -17.84, 46.554] deg; flange x=-566.205 y=-22.511 z=329.267 mm, rx=1.5153 ry=-0.5827 rz=0.5877 rad
    Loop Counting (count=1) loopVariable(name=Loop_8)
      MoveP speed 38.1 mm/s, acceleration 17.78 mm/s^2 (blendRadius=0.0127 recalculateMotions=false) feature=Base
        CircleMove
          Waypoint Waypoint_74: TCP in base x=-581.748 y=-232.335 z=325.131 mm, rx=0.6953 ry=1.8078 rz=-1.7617 rad; joints [-14.981, -64.989, 72.108, -11.678, -15.633, 47.126] deg; flange x=-583.981 y=-40.283 z=329.284 mm, rx=1.5154 ry=-0.5825 rz=0.5876 rad
          Waypoint Waypoint_75: TCP in base x=-600.204 y=-216.337 z=325.252 mm, rx=0.6933 ry=1.8095 rz=-1.7634 rad; joints [-16.013, -62.061, 67.737, -9.96, -16.653, 46.7] deg; flange x=-602.441 y=-24.235 z=329.378 mm, rx=1.5158 ry=-0.5807 rz=0.5857 rad
        CircleMove
          Waypoint Waypoint_76: TCP in base x=-582.7 y=-198.306 z=325.197 mm, rx=0.6964 ry=1.807 rz=-1.7609 rad; joints [-18.188, -64.188, 70.919, -10.531, -18.821, 46.417] deg; flange x=-584.928 y=-6.239 z=329.276 mm, rx=1.515 ry=-0.5838 rz=0.5887 rad
          Waypoint Waypoint_77: TCP in base x=-564.342 y=-207.565 z=325.189 mm, rx=0.6953 ry=1.8079 rz=-1.7618 rad; joints [-17.882, -66.961, 74.945, -11.84, -18.513, 46.402] deg; flange x=-566.548 y=-15.408 z=329.285 mm, rx=1.5152 ry=-0.5828 rz=0.5876 rad
    MoveP speed 25.4 mm/s, acceleration 7.62 mm/s^2 (blendRadius=0.00762 recalculateMotions=false) feature=Base
      CircleMove
        Waypoint Waypoint_78: TCP in base x=-581.791 y=-232.277 z=325.145 mm, rx=0.6954 ry=1.8079 rz=-1.7618 rad; joints [-14.988, -64.985, 72.111, -11.674, -15.633, 47.129] deg; flange x=-583.987 y=-40.212 z=329.219 mm, rx=1.5152 ry=-0.5828 rz=0.5878 rad
        Waypoint Waypoint_79: TCP in base x=-600.181 y=-216.355 z=325.262 mm, rx=0.6932 ry=1.8096 rz=-1.7634 rad; joints [-16.015, -62.061, 67.741, -9.962, -16.655, 46.7] deg; flange x=-602.438 y=-24.214 z=329.348 mm, rx=1.5158 ry=-0.5807 rz=0.5857 rad
      CircleMove
        Waypoint Waypoint_80: TCP in base x=-587.826 y=-205.303 z=325.197 mm, rx=0.6955 ry=1.8076 rz=-1.7617 rad; joints [-17.381, -63.614, 70.068, -10.411, -18.017, 46.515] deg; flange x=-590.045 y=-13.224 z=329.31 mm, rx=1.5152 ry=-0.5828 rz=0.5878 rad
        Waypoint next_47: TCP in base x=-579.353 y=-207.539 z=325.273 mm, rx=0.7058 ry=1.7993 rz=-1.7532 rad; joints [-17.422, -64.869, 71.912, -11.004, -18.052, 47.285] deg; flange x=-581.56 y=-15.439 z=329.346 mm, rx=1.5123 ry=-0.5935 rz=0.5979 rad
    Waypoint cent_47: motionParameters(blendRadius=0); TCP in base x=-579.349 y=-207.563 z=325.249 mm, rx=0.706 ry=1.7991 rz=-1.7531 rad; joints [-17.42, -64.861, 71.913, -11, -18.052, 47.287] deg; flange x=-581.58 y=-15.454 z=329.264 mm, rx=1.5122 ry=-0.5936 rz=0.5982 rad
    Loop Counting (count=1) loopVariable(name=Loop_9)
      MoveP speed 25.4 mm/s, acceleration 25.4 mm/s^2 (blendRadius=0.00762 recalculateMotions=false) feature=Base
        CircleMove
          Waypoint Waypoint_81: TCP in base x=-588.1 y=-215.124 z=325.198 mm, rx=0.7063 ry=1.7987 rz=-1.7529 rad; joints [-16.453, -63.777, 70.316, -10.706, -17.084, 47.514] deg; flange x=-590.334 y=-23.032 z=329.289 mm, rx=1.5122 ry=-0.5936 rz=0.5981 rad
          Waypoint Waypoint_82: TCP in base x=-595.697 y=-207.572 z=325.287 mm, rx=0.706 ry=1.7991 rz=-1.753 rad; joints [-16.949, -62.534, 68.449, -9.978, -17.585, 47.394] deg; flange x=-597.935 y=-15.437 z=329.349 mm, rx=1.5124 ry=-0.5935 rz=0.598 rad
        CircleMove
          Waypoint Waypoint_83: TCP in base x=-585.259 y=-202.778 z=325.22 mm, rx=0.7063 ry=1.7988 rz=-1.753 rad; joints [-17.696, -63.931, 70.538, -10.504, -18.324, 47.227] deg; flange x=-587.449 y=-10.681 z=329.294 mm, rx=1.5122 ry=-0.5936 rz=0.5981 rad
          Waypoint Waypoint_84: TCP in base x=-579.374 y=-207.55 z=325.181 mm, rx=0.7061 ry=1.7989 rz=-1.753 rad; joints [-17.42, -64.861, 71.913, -11, -18.052, 47.287] deg; flange x=-581.58 y=-15.454 z=329.264 mm, rx=1.5122 ry=-0.5936 rz=0.5982 rad
    MoveP speed 25.4 mm/s, acceleration 12.7 mm/s^2 (blendRadius=0.00762 recalculateMotions=false) feature=Base
      CircleMove
        Waypoint Waypoint_85: TCP in base x=-588.1 y=-215.124 z=325.198 mm, rx=0.7063 ry=1.7987 rz=-1.7529 rad; joints [-16.453, -63.777, 70.316, -10.706, -17.084, 47.514] deg; flange x=-590.334 y=-23.032 z=329.289 mm, rx=1.5122 ry=-0.5936 rz=0.5981 rad
        Waypoint Waypoint_86: TCP in base x=-595.697 y=-207.572 z=325.287 mm, rx=0.706 ry=1.7991 rz=-1.753 rad; joints [-16.949, -62.534, 68.449, -9.978, -17.585, 47.394] deg; flange x=-597.935 y=-15.437 z=329.349 mm, rx=1.5124 ry=-0.5935 rz=0.598 rad
      CircleMove
        Waypoint Waypoint_87: motionParameters(jointSpeed=1.047198 jointAcceleration=1.396263 cartesianSpeed=0.02032 cartesianAcceleration=0.02286); TCP in base x=-585.259 y=-202.778 z=325.22 mm, rx=0.7063 ry=1.7988 rz=-1.753 rad; joints [-17.696, -63.931, 70.538, -10.504, -18.324, 47.227] deg; flange x=-587.449 y=-10.681 z=329.294 mm, rx=1.5122 ry=-0.5936 rz=0.5981 rad
        Waypoint next_48: TCP in base x=-581.585 y=-207.501 z=326.28 mm, rx=0.7198 ry=1.7875 rz=-1.7417 rad; joints [-17.362, -64.57, 71.32, -10.723, -17.986, 48.303] deg; flange x=-583.802 y=-15.379 z=330.384 mm, rx=1.5084 ry=-0.6074 rz=0.6114 rad
    Waypoint cent_48: motionParameters(blendRadius=0); TCP in base x=-581.612 y=-207.503 z=326.29 mm, rx=0.7198 ry=1.7876 rz=-1.7418 rad; joints [-17.357, -64.57, 71.319, -10.72, -17.987, 48.299] deg; flange x=-583.793 y=-15.428 z=330.399 mm, rx=1.5085 ry=-0.6073 rz=0.6114 rad
    Loop Counting (count=1) loopVariable(name=Loop_10)
      MoveP speed 25.4 mm/s, acceleration 7.62 mm/s^2 (blendRadius=0.00762 recalculateMotions=false) feature=Base
        CircleMove
          Waypoint Waypoint_88: TCP in base x=-589.206 y=-215.124 z=326.256 mm, rx=0.7199 ry=1.7874 rz=-1.7417 rad; joints [-16.425, -63.64, 69.954, -10.494, -17.051, 48.524] deg; flange x=-591.427 y=-23.005 z=330.372 mm, rx=1.5084 ry=-0.6074 rz=0.6114 rad
          Waypoint Waypoint_89: TCP in base x=-596.831 y=-207.448 z=326.349 mm, rx=0.7198 ry=1.7877 rz=-1.7418 rad; joints [-16.929, -62.395, 68.079, -9.764, -17.552, 48.405] deg; flange x=-599.032 y=-15.332 z=330.447 mm, rx=1.5085 ry=-0.6073 rz=0.6112 rad
        CircleMove
          Waypoint Waypoint_90: TCP in base x=-589.25 y=-199.746 z=326.33 mm, rx=0.7198 ry=1.7879 rz=-1.742 rad; joints [-17.857, -63.323, 69.465, -10.026, -18.473, 48.192] deg; flange x=-591.425 y=-7.689 z=330.444 mm, rx=1.5085 ry=-0.6073 rz=0.611 rad
          Waypoint Waypoint_91: TCP in base x=-581.603 y=-207.512 z=326.29 mm, rx=0.7198 ry=1.7875 rz=-1.7417 rad; joints [-17.357, -64.57, 71.319, -10.72, -17.987, 48.299] deg; flange x=-583.793 y=-15.428 z=330.399 mm, rx=1.5085 ry=-0.6073 rz=0.6114 rad
    MoveP speed 25.4 mm/s, acceleration 12.7 mm/s^2 (blendRadius=0.00889 recalculateMotions=false) feature=Base
      CircleMove
        Waypoint Waypoint_92: TCP in base x=-589.206 y=-215.124 z=326.256 mm, rx=0.7199 ry=1.7874 rz=-1.7417 rad; joints [-16.425, -63.64, 69.954, -10.494, -17.051, 48.524] deg; flange x=-591.427 y=-23.005 z=330.372 mm, rx=1.5084 ry=-0.6074 rz=0.6114 rad
        Waypoint Waypoint_93: motionParameters(blendRadius=0.007024); TCP in base x=-603.981 y=-207.404 z=326.377 mm, rx=0.7199 ry=1.7877 rz=-1.7419 rad; joints [-16.732, -61.358, 66.509, -9.275, -17.354, 48.454] deg; flange x=-606.159 y=-15.324 z=330.456 mm, rx=1.5085 ry=-0.6074 rz=0.6112 rad
      CircleMove
        Waypoint Waypoint_94: motionParameters(jointSpeed=1.047198 jointAcceleration=1.396263 cartesianSpeed=0.02286 cartesianAcceleration=0.0254 blendRadius=0.003002); TCP in base x=-589.275 y=-199.747 z=326.305 mm, rx=0.7197 ry=1.7879 rz=-1.7421 rad; joints [-17.864, -63.324, 69.469, -10.026, -18.477, 48.19] deg; flange x=-591.406 y=-7.622 z=330.438 mm, rx=1.5085 ry=-0.6073 rz=0.611 rad
        Waypoint next_49: motionParameters(jointSpeed=1.047198 jointAcceleration=1.396263 cartesianSpeed=0.02032 cartesianAcceleration=0.0254); TCP in base x=-578.891 y=-207.506 z=326.331 mm, rx=0.7327 ry=1.7767 rz=-1.7309 rad; joints [-17.441, -64.95, 71.878, -10.88, -18.066, 49.243] deg; flange x=-581.102 y=-15.388 z=330.381 mm, rx=1.5046 ry=-0.6205 rz=0.6242 rad
    Loop Counting (count=1) loopVariable(name=Loop_11)
      MoveP speed 33.02 mm/s, acceleration 17.78 mm/s^2 (blendRadius=0.0254 recalculateMotions=false) feature=Base
        CircleMove
          Waypoint Waypoint_95: TCP in base x=-593.528 y=-232.87 z=333.329 mm, rx=0.7318 ry=1.7774 rz=-1.7315 rad; joints [-14.642, -63.448, 68.641, -9.857, -15.275, 49.921] deg; flange x=-595.746 y=-40.752 z=337.418 mm, rx=1.5049 ry=-0.6197 rz=0.6234 rad
          Waypoint Waypoint_96: TCP in base x=-616.939 y=-211.212 z=337.96 mm, rx=0.7316 ry=1.7774 rz=-1.7314 rad; joints [-16.046, -59.602, 62.117, -6.792, -16.686, 49.511] deg; flange x=-619.194 y=-19.075 z=342.059 mm, rx=1.5051 ry=-0.6195 rz=0.6234 rad
        CircleMove
          Waypoint Waypoint_97: TCP in base x=-591.5 y=-185.807 z=337.994 mm, rx=0.7314 ry=1.7776 rz=-1.7315 rad; joints [-19.077, -62.79, 66.954, -7.806, -19.714, 48.842] deg; flange x=-593.769 y=6.323 z=342.115 mm, rx=1.5051 ry=-0.6194 rz=0.6234 rad
          Waypoint Waypoint_98: TCP in base x=-568.091 y=-207.558 z=327.452 mm, rx=0.7317 ry=1.7775 rz=-1.7315 rad; joints [-17.764, -66.489, 73.932, -11.338, -18.397, 49.117] deg; flange x=-570.284 y=-15.434 z=331.569 mm, rx=1.505 ry=-0.6196 rz=0.6235 rad
    MoveP speed 33.02 mm/s, acceleration 12.7 mm/s^2 (blendRadius=0.00762 recalculateMotions=false) feature=Base
      CircleMove
        Waypoint Waypoint_99: TCP in base x=-593.509 y=-232.895 z=329.334 mm, rx=0.7318 ry=1.7774 rz=-1.7315 rad; joints [-14.644, -63.398, 69.15, -10.413, -15.277, 49.922] deg; flange x=-595.705 y=-40.741 z=333.455 mm, rx=1.5049 ry=-0.6197 rz=0.6234 rad
        Waypoint Waypoint_100: TCP in base x=-596.757 y=-207.583 z=327.474 mm, rx=0.7317 ry=1.7774 rz=-1.7316 rad; joints [-16.921, -62.414, 67.944, -9.605, -17.552, 49.296] deg; flange x=-599 y=-15.419 z=331.567 mm, rx=1.505 ry=-0.6195 rz=0.6233 rad
      CircleMove
        Waypoint Waypoint_101: motionParameters(blendRadius=0.002); TCP in base x=-589.178 y=-199.893 z=327.487 mm, rx=0.7317 ry=1.7776 rz=-1.7316 rad; joints [-17.847, -63.343, 69.328, -9.87, -18.477, 49.095] deg; flange x=-591.401 y=-7.792 z=331.579 mm, rx=1.5051 ry=-0.6195 rz=0.6233 rad
        Waypoint next_50: TCP in base x=-580.743 y=-214.605 z=329.493 mm, rx=0.745 ry=1.7663 rz=-1.7202 rad; joints [-16.713, -64.892, 71.316, -10.575, -17.345, 50.359] deg; flange x=-582.975 y=-22.469 z=333.637 mm, rx=1.5012 ry=-0.6331 rz=0.6364 rad
    Waypoint cent_50: motionParameters(blendRadius=0); TCP in base x=-580.768 y=-214.592 z=329.504 mm, rx=0.7449 ry=1.7664 rz=-1.7203 rad; joints [-16.713, -64.888, 71.316, -10.569, -17.34, 50.358] deg; flange x=-582.988 y=-22.464 z=333.595 mm, rx=1.5011 ry=-0.6332 rz=0.6365 rad
    Loop Counting (count=2) loopVariable(name=Loop_12)
      MoveP speed 35.56 mm/s, acceleration 12.7 mm/s^2 (blendRadius=0.00762 recalculateMotions=false) feature=Base
        CircleMove
          Waypoint Waypoint_102: TCP in base x=-599.806 y=-233.683 z=335.12 mm, rx=0.745 ry=1.7663 rz=-1.7202 rad; joints [-14.419, -62.579, 67.076, -9.26, -15.05, 50.998] deg; flange x=-602.019 y=-41.51 z=339.251 mm, rx=1.5011 ry=-0.6332 rz=0.6364 rad
          Waypoint Waypoint_103: TCP in base x=-617.512 y=-215.323 z=347.306 mm, rx=0.7448 ry=1.7665 rz=-1.7203 rad; joints [-15.659, -59.661, 60.844, -5.585, -16.293, 50.619] deg; flange x=-619.743 y=-23.23 z=351.398 mm, rx=1.5012 ry=-0.6331 rz=0.6364 rad
        CircleMove
          Waypoint Waypoint_104: TCP in base x=-598.385 y=-196.328 z=347.37 mm, rx=0.7446 ry=1.7666 rz=-1.7203 rad; joints [-17.907, -62.129, 64.594, -6.352, -18.538, 50.078] deg; flange x=-600.638 y=-4.175 z=351.464 mm, rx=1.5012 ry=-0.633 rz=0.6364 rad
          Waypoint Waypoint_105: TCP in base x=-580.753 y=-214.638 z=329.55 mm, rx=0.7449 ry=1.7664 rz=-1.7203 rad; joints [-16.713, -64.892, 71.316, -10.575, -17.345, 50.359] deg; flange x=-582.975 y=-22.469 z=333.637 mm, rx=1.5012 ry=-0.6331 rz=0.6364 rad
    MoveP speed 25.4 mm/s, acceleration 12.7 mm/s^2 (blendRadius=0.00762 recalculateMotions=false) feature=Base
      CircleMove
        Waypoint Waypoint_106: TCP in base x=-599.794 y=-233.68 z=335.119 mm, rx=0.745 ry=1.7663 rz=-1.7202 rad; joints [-14.415, -62.58, 67.076, -9.259, -15.052, 51.002] deg; flange x=-602.01 y=-41.56 z=339.252 mm, rx=1.5012 ry=-0.6332 rz=0.6365 rad
        Waypoint Waypoint_107: TCP in base x=-617.457 y=-215.332 z=347.324 mm, rx=0.7447 ry=1.7665 rz=-1.7203 rad; joints [-15.662, -59.665, 60.842, -5.586, -16.299, 50.621] deg; flange x=-619.722 y=-23.2 z=351.445 mm, rx=1.5013 ry=-0.633 rz=0.6364 rad
      CircleMove
        Waypoint Waypoint_108: motionParameters(blendRadius=0); TCP in base x=-589.134 y=-199.873 z=329.43 mm, rx=0.745 ry=1.7663 rz=-1.7203 rad; joints [-17.855, -63.379, 69.096, -9.609, -18.48, 50.1] deg; flange x=-591.359 y=-7.727 z=333.524 mm, rx=1.5011 ry=-0.6333 rz=0.6366 rad
        Waypoint next_51: TCP in base x=-590.05 y=-208.06 z=331.987 mm, rx=0.757 ry=1.7559 rz=-1.7101 rad; joints [-17.063, -63.473, 68.859, -9.445, -17.691, 51.167] deg; flange x=-592.214 y=-15.963 z=336.113 mm, rx=1.4974 ry=-0.6455 rz=0.6485 rad
    Waypoint cent_51: motionParameters(blendRadius=0); TCP in base x=-590.016 y=-208.087 z=331.992 mm, rx=0.7569 ry=1.7559 rz=-1.7101 rad; joints [-17.064, -63.475, 68.86, -9.448, -17.691, 51.168] deg; flange x=-592.21 y=-15.95 z=336.122 mm, rx=1.4974 ry=-0.6455 rz=0.6484 rad
    Loop Counting (count=2) loopVariable(name=Loop_13)
      MoveP speed 38.1 mm/s, acceleration 7.62 mm/s^2 (blendRadius=0.00762 recalculateMotions=false) feature=Base
        CircleMove
          Waypoint Waypoint_109: TCP in base x=-597.659 y=-215.648 z=331.967 mm, rx=0.7571 ry=1.7558 rz=-1.7101 rad; joints [-16.142, -62.525, 67.45, -9.199, -16.774, 51.393] deg; flange x=-599.836 y=-23.589 z=336.086 mm, rx=1.4974 ry=-0.6455 rz=0.6485 rad
          Waypoint Waypoint_110: TCP in base x=-605.201 y=-208.051 z=332.02 mm, rx=0.7571 ry=1.7557 rz=-1.71 rad; joints [-16.643, -61.254, 65.522, -8.419, -17.267, 51.272] deg; flange x=-607.428 y=-15.924 z=336.108 mm, rx=1.4973 ry=-0.6456 rz=0.6486 rad
        CircleMove
          Waypoint Waypoint_111: TCP in base x=-597.626 y=-200.297 z=331.916 mm, rx=0.7571 ry=1.7557 rz=-1.7099 rad; joints [-17.559, -62.199, 66.959, -8.703, -18.183, 51.062] deg; flange x=-599.814 y=-8.242 z=336.05 mm, rx=1.4973 ry=-0.6457 rz=0.6487 rad
          Waypoint Waypoint_112: TCP in base x=-590.05 y=-208.081 z=331.961 mm, rx=0.757 ry=1.7558 rz=-1.71 rad; joints [-17.063, -63.473, 68.859, -9.445, -17.691, 51.167] deg; flange x=-592.214 y=-15.963 z=336.113 mm, rx=1.4974 ry=-0.6455 rz=0.6485 rad
    MoveP speed 25.4 mm/s, acceleration 12.7 mm/s^2 (blendRadius=0.00762 recalculateMotions=false) feature=Base
      CircleMove
        Waypoint Waypoint_113: TCP in base x=-589.917 y=-215.126 z=332.051 mm, rx=0.7566 ry=1.7563 rz=-1.7102 rad; joints [-16.401, -63.632, 69.092, -9.679, -17.03, 51.331] deg; flange x=-592.139 y=-23.05 z=336.144 mm, rx=1.4975 ry=-0.6455 rz=0.6484 rad
        Waypoint Waypoint_114: TCP in base x=-597.485 y=-207.562 z=332.048 mm, rx=0.7567 ry=1.7561 rz=-1.71 rad; joints [-16.899, -62.372, 67.208, -8.945, -17.535, 51.207] deg; flange x=-599.749 y=-15.429 z=336.145 mm, rx=1.4976 ry=-0.6453 rz=0.6484 rad
      CircleMove
        Waypoint Waypoint_115: motionParameters(blendRadius=0.002); TCP in base x=-589.923 y=-199.93 z=332.01 mm, rx=0.7566 ry=1.7563 rz=-1.7103 rad; joints [-17.828, -63.307, 68.605, -9.206, -18.449, 50.992] deg; flange x=-592.146 y=-7.767 z=336.133 mm, rx=1.4975 ry=-0.6454 rz=0.6482 rad
        Waypoint next_52: motionParameters(jointSpeed=1.047198 jointAcceleration=1.396263 cartesianSpeed=0.01778 cartesianAcceleration=0.0254); TCP in base x=-582.293 y=-207.503 z=331.968 mm, rx=0.7726 ry=1.742 rz=-1.6963 rad; joints [-17.342, -64.561, 70.472, -9.903, -17.967, 52.295] deg; flange x=-584.515 y=-15.367 z=336.067 mm, rx=1.4923 ry=-0.6619 rz=0.6645 rad
    Waypoint cent_52: motionParameters(blendRadius=0); TCP in base x=-596.115 y=-207.466 z=331.995 mm, rx=0.7726 ry=1.7421 rz=-1.6965 rad; joints [-16.946, -62.578, 67.53, -9.03, -17.572, 52.385] deg; flange x=-598.296 y=-15.367 z=336.067 mm, rx=1.4923 ry=-0.6619 rz=0.6645 rad
    MoveP speed 25.4 mm/s, acceleration 7.62 mm/s^2 (blendRadius=0.00635 recalculateMotions=false) feature=Base
      CircleMove
        Waypoint Waypoint_116: TCP in base x=-602.421 y=-213.729 z=332.011 mm, rx=0.7725 ry=1.7422 rz=-1.6966 rad; joints [-16.191, -61.789, 66.335, -8.809, -16.817, 52.563] deg; flange x=-604.619 y=-21.681 z=336.118 mm, rx=1.4924 ry=-0.6617 rz=0.6643 rad
        Waypoint Waypoint_117: TCP in base x=-608.78 y=-207.464 z=335.305 mm, rx=0.7724 ry=1.7422 rz=-1.6966 rad; joints [-16.6, -60.749, 64.266, -7.681, -17.225, 52.459] deg; flange x=-610.971 y=-15.338 z=339.419 mm, rx=1.4924 ry=-0.6617 rz=0.6643 rad
      CircleMove
        Waypoint Waypoint_118: TCP in base x=-602.419 y=-201.11 z=335.281 mm, rx=0.7723 ry=1.7423 rz=-1.6965 rad; joints [-17.354, -61.553, 65.487, -7.931, -17.977, 52.28] deg; flange x=-604.609 y=-8.977 z=339.43 mm, rx=1.4924 ry=-0.6617 rz=0.6642 rad
        Waypoint Waypoint_119: motionParameters(jointSpeed=1.047198 jointAcceleration=1.396263 cartesianSpeed=0.01778 cartesianAcceleration=0.0254); TCP in base x=-596.13 y=-207.493 z=331.982 mm, rx=0.7726 ry=1.7421 rz=-1.6966 rad; joints [-16.949, -62.582, 67.528, -9.028, -17.569, 52.38] deg; flange x=-598.288 y=-15.342 z=336.11 mm, rx=1.4923 ry=-0.6619 rz=0.6643 rad
    Wait Sleep waitTime=0.5
  MoveL speed 76.2 mm/s, acceleration 635 mm/s^2 (recalculateMotions=false) feature=Base
    Waypoint cup_cent: TCP in base x=-571.578 y=-210.276 z=318.459 mm, rx=0.4644 ry=1.9797 rz=-1.9328 rad; joints [-17.399, -65.896, 74.417, -12.484, -18.002, 30.817] deg; flange x=-573.709 y=-18.152 z=322.504 mm, rx=1.5623 ry=-0.3665 rz=0.3757 rad
  Wait Sleep waitTime=10
  MoveL speed 101.6 mm/s, acceleration 889 mm/s^2 (recalculateMotions=false) feature=Base
    Waypoint Waypoint_13: TCP in base x=-258.775 y=-200.368 z=296.07 mm, rx=0.373 ry=1.9901 rz=-1.9468 rad; joints [-37.125, -106.526, 121.704, -16.151, -40.089, 24.993] deg; flange x=-268.58 y=-13.971 z=298.092 mm, rx=1.5665 ry=-0.2937 rz=0.3713 rad
    Waypoint putdown: TCP in base x=-228.919 y=-202.017 z=57.158 mm, rx=0.3489 ry=2.0764 rz=-2.0657 rad; joints [-45.414, -84.511, 150.263, -66.622, -43.64, 18.05] deg; flange x=-223.324 y=-15.473 z=58.966 mm, rx=1.5625 ry=-0.2627 rz=0.2138 rad
    URCap com.ur.urcap.OnRobot.HelloWorldNode data=depthCompensate = false
      | width = 40
      | name = RG2(40)
      | force = 40
  MoveJ speed 40 deg/s, acceleration 60 deg/s^2 (recalculateMotions=false)
    Waypoint Waypoint_4: TCP in base x=-230.104 y=-131.648 z=57.167 mm, rx=0.3489 ry=2.0764 rz=-2.0657 rad; joints [-57.471, -80.568, 144.978, -65.128, -55.694, 17.825] deg; flange x=-224.374 y=60.451 z=59.028 mm, rx=1.5626 ry=-0.2626 rz=0.2137 rad
    Waypoint Waypoint_23: TCP in base x=-760.946 y=131.205 z=228.784 mm, rx=-1.536 ry=-0.9541 rz=1.6135 rad; joints [-28.947, -70.668, 96.865, -27.78, 58.701, 29.555] deg; flange x=-568.994 y=139.38 z=224.143 mm, rx=0.8464 ry=-1.3627 rz=-0.8068 rad
    Waypoint Waypoint_1: TCP in base x=-743.769 y=-4.694 z=207.878 mm, rx=-1.1781 ry=-1.2348 rz=1.2992 rad; joints [-15.586, -73.845, 104.669, -32.199, 70.077, 2.173] deg; flange x=-552.191 y=10.079 z=203.405 mm, rx=1.2063 ry=-1.1509 rz=-1.1399 rad
    Waypoint Waypoint_20: TCP in base x=-692.574 y=-209.421 z=156.932 mm, rx=-1.178 ry=-1.2351 rz=1.2993 rad; joints [10.29, -71.059, 109.838, -40.098, 95.938, 1.547] deg; flange x=-501.03 y=-194.617 z=152.52 mm, rx=1.2063 ry=-1.1506 rz=-1.1399 rad
    URCap com.ur.urcap.OnRobot.HelloWorldNode data=depthCompensate = false
      | width = 90
      | name = RG2(90)
      | force = 40
      | payload = 0.0
  MoveL speed 76.2 mm/s, acceleration 635 mm/s^2 (recalculateMotions=false) feature=Base
    Waypoint Waypoint_12: motionParameters(jointSpeed=1.047198 jointAcceleration=1.396263 cartesianSpeed=0.127 cartesianAcceleration=0.508); TCP in base x=-788.554 y=-209.398 z=154.524 mm, rx=-1.178 ry=-1.2351 rz=1.2992 rad; joints [8.457, -60.699, 94.236, -34.85, 94.112, 1.593] deg; flange x=-597.005 y=-194.617 z=150.12 mm, rx=1.2063 ry=-1.1506 rz=-1.1399 rad
    Waypoint Waypoint_15: motionParameters(jointSpeed=1.047198 jointAcceleration=1.396263 cartesianSpeed=0.0254 cartesianAcceleration=0.254); TCP in base x=-836.88 y=-209.476 z=144.361 mm, rx=-1.1779 ry=-1.2352 rz=1.2993 rad; joints [7.755, -54.667, 85.83, -32.474, 93.414, 1.609] deg; flange x=-645.319 y=-194.617 z=139.949 mm, rx=1.2063 ry=-1.1506 rz=-1.1399 rad
    URCap com.ur.urcap.OnRobot.HelloWorldNode data=depthCompensate = false
      | width = 0
      | name = RG2(0)
      | force = 40
    Waypoint Waypoint_16: TCP in base x=-836.872 y=-209.404 z=165.163 mm, rx=-1.178 ry=-1.2351 rz=1.2993 rad; joints [7.756, -56.07, 84.724, -29.966, 93.413, 1.612] deg; flange x=-645.319 y=-194.617 z=160.732 mm, rx=1.2063 ry=-1.1506 rz=-1.1399 rad
    Waypoint Waypoint_17: motionParameters(jointSpeed=1.047198 jointAcceleration=1.396263 cartesianSpeed=0.0762 cartesianAcceleration=0.254); TCP in base x=-833.298 y=-44.185 z=165.184 mm, rx=-1.1781 ry=-1.235 rz=1.2993 rad; joints [-9.026, -60.089, 91.399, -32.648, 76.637, 2.004] deg; flange x=-641.753 y=-29.398 z=160.753 mm, rx=1.2063 ry=-1.1506 rz=-1.1399 rad
    Waypoint Waypoint_21: motionParameters(jointSpeed=1.047198 jointAcceleration=1.396263 cartesianSpeed=0.0254 cartesianAcceleration=0.254); TCP in base x=-833.333 y=-44.187 z=108.239 mm, rx=-1.1778 ry=-1.235 rz=1.2993 rad; joints [-9.032, -55.694, 94.064, -39.714, 76.636, 1.987] deg; flange x=-641.776 y=-29.36 z=103.821 mm, rx=1.2063 ry=-1.1505 rz=-1.1401 rad
    URCap com.ur.urcap.OnRobot.HelloWorldNode data=depthCompensate = false
      | width = 90
      | name = RG2(90)
      | force = 40
    Waypoint Waypoint_18: motionParameters(jointSpeed=1.047198 jointAcceleration=1.396263 cartesianSpeed=0.0508 cartesianAcceleration=0.508); TCP in base x=-722.466 y=-41.748 z=104.2 mm, rx=-1.178 ry=-1.2351 rz=1.2993 rad; joints [-11.615, -66.927, 114.057, -48.478, 74.042, 2.046] deg; flange x=-530.936 y=-26.926 z=99.754 mm, rx=1.2063 ry=-1.1506 rz=-1.1399 rad
    MoveJ speed 40 deg/s, acceleration 50 deg/s^2 (recalculateMotions=false)
      Waypoint Waypoint_19: motionParameters(jointSpeed=1.047198 jointAcceleration=1.396263 cartesianSpeed=0.1778 cartesianAcceleration=1.2); TCP in base x=-622.981 y=-125.831 z=100.302 mm, rx=-0.6658 ry=-1.814 rz=1.8405 rad; joints [-24.893, -66.198, 112.873, -48.51, 14.605, 2.663] deg; flange x=-500.966 y=22.628 z=98.59 mm, rx=1.4892 ry=-0.5465 rz=-0.5279 rad
      Waypoint Waypoint_22: motionParameters(nextMotionTime=3); TCP in base x=-485.513 y=-120.248 z=100.265 mm, rx=-0.6659 ry=-1.8141 rz=1.8407 rad; joints [-36.356, -81.603, 135.743, -62.436, 3.163, 9.179] deg; flange x=-363.542 y=28.228 z=98.59 mm, rx=1.4892 ry=-0.5465 rz=-0.5279 rad
      URCap com.ur.urcap.OnRobot.HelloWorldNode data=depthCompensate = false
        | width = 20
        | name = RG2(20)
        | force = 40
      Waypoint Waypoint_25: motionParameters(jointSpeed=1.047198 jointAcceleration=1.396263 cartesianSpeed=0.249758 cartesianAcceleration=1.2); TCP in base x=-274.75 y=-2.206 z=93.829 mm, rx=0.6697 ry=1.7766 rz=-1.859 rad; joints [-61.662, -71.825, 125.124, -50.852, -60.403, 38.941] deg; flange x=-270.843 y=184.262 z=86.813 mm, rx=1.4577 ry=-0.5495 rz=0.5386 rad
